(*			
	RafalOS
	Rafał Osajda		20.11.2025		TC 4024.66
	Moduł przygotowania danych dla Okna parametrów we wsztsystkich trybach
*)
FUNCTION_BLOCK FB_MCHMIPrepareDataForScreen_01_XX EXTENDS FB_MCHMIPrepareDataForScreen IMPLEMENTS ITF_MCHMIPrepareDataForScreen
VAR
	itfMachineControlHMI	: ITF_MCHMIMachineControl_HMI_PrepScr_01_XX;
	refstData				: REFERENCE TO ST_MCHMIPrepareScreen_01_XX;
END_VAR

(*			
	RafalOS
	Rafał Osajda		19.11.2025		TC 4024.66
	Czyści danych przy zmienia ramki po poprzedniej ramce
*)
METHOD PUBLIC ClearAfterScreen : BOOL
VAR_INPUT
END_VAR
SUPER^.ClearAfterScreen ();
END_METHOD

METHOD PRIVATE CreateListName
VAR_INPUT
END_VAR
END_METHOD

METHOD PUBLIC LinkDataHMI_01_XX : BOOL
VAR_INPUT
	refstData				: REFERENCE TO ST_MCHMIPrepareScreen_01_XX;
END_VAR
THIS^.refstData REF= refstData;
END_METHOD

METHOD PUBLIC LinkMachineControlHMI : BOOL
VAR_INPUT
	fbMachineControlHMI	: ITF_MCHMIMachineControl_HMI_PrepScr_01_XX;
END_VAR
this^.itfMachineControlHMI := fbMachineControlHMI;
END_METHOD

(*			
	RafalOS
	Rafał Osajda		14.11.2025		TC 4024.66
	Metoda przygotowywania danych dla HMI 
	W niej odbywa się odpytywanie właściego elementu przez łącznik
*)
METHOD PUBLIC PrepareDataForHMI : BOOL
VAR_INPUT
END_VAR

IF (THIS^.refstHMICommonData.bChangePage) THEN
	THIS^.CreateListName ();
END_IF





SUPER^.PrepareDataForHMI ();
END_METHOD

(*			
	RafalOS
	Rafał Osajda		19.11.2025		TC 4024.66
	Przygotowanie ramki pood tamke do wyświetlenia - tylko przygotowanie a nie przygotowanie danych do wyświetlenia
*)
METHOD PUBLIC PrepareForScreen : BOOL
VAR_INPUT
END_VAR
SUPER^.PrepareForScreen ();
END_METHOD

END_FUNCTION_BLOCK

(* stored: Version 1.1.0.1
   POU FB_MCHMIPrepareDataForScreen_01_XX: Id {62188713-537e-0ba6-3aee-7a017ce7ab57}, SpecialFunc None
   Folder ITF_PDFS: Id {88be56d6-550f-028a-26d5-d43e2e2a4238}
   Method ClearAfterScreen: Id {a8c50998-1268-0361-3361-f40b48e5bd11}
   Method CreateListName: Id {dfb83b60-14e0-0020-26db-362d83675795}
   Method LinkDataHMI_01_XX: Id {0241f470-6f5d-05e7-0457-a5cdb3f66823}
   Method LinkMachineControlHMI: Id {be4941eb-3101-0648-3fed-d300417ecd90}
   Method PrepareDataForHMI: Id {4067778e-275e-044f-0fd9-c3f95f0c4867}
   Method PrepareForScreen: Id {af3a1d4b-6467-08de-039f-018bb4326fe0} *)
